FUNCTION_BLOCK FB_CloseIO
VAR_INPUT
END_VAR
VAR_OUTPUT
END_VAR
VAR
	idx				: INT:=1;
	CloseAir			: FB_CloseAir;
	CloseOil			: FB_CloseOil;
END_VAR

FOR idx:=1 TO TouchNo DO
	Touch[idx].CurTime := 0;
END_FOR

CloseAir();

CloseOil();

END_FUNCTION_BLOCK

(* stored: Version 1.1.0.1, ProductVersion 3.1.4024.9
   POU FB_CloseIO: Id {85e66412-8b54-4367-86fb-f00f9f1f2bad}, SpecialFunc None *)
